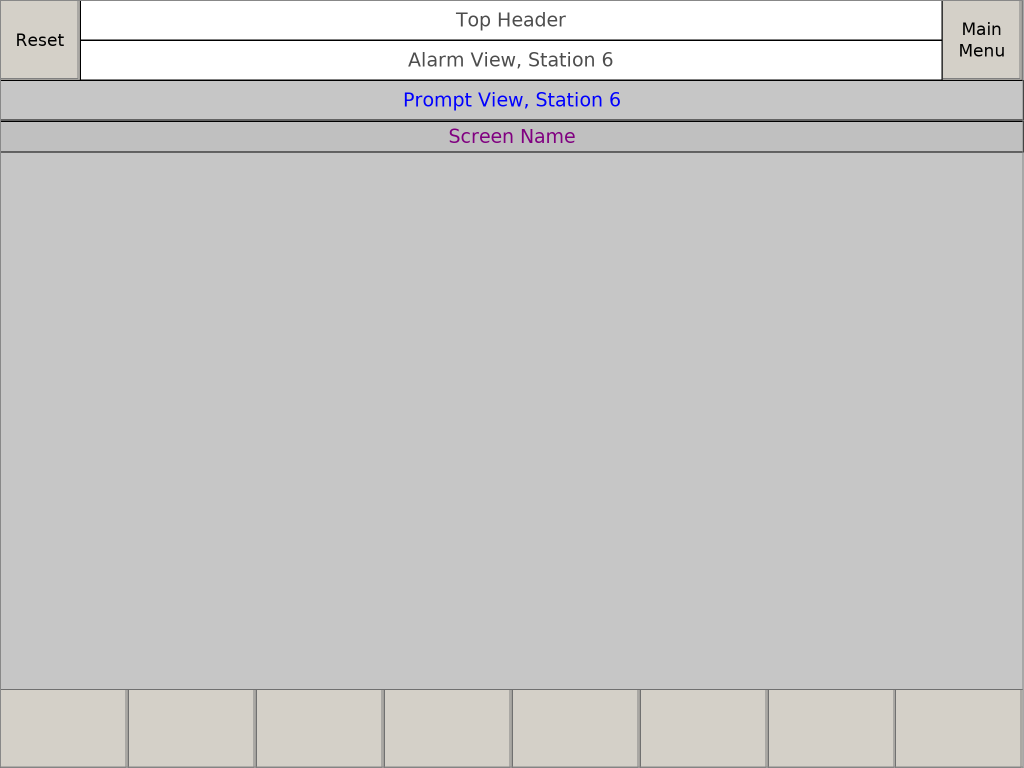
VISUALIZATION SS_91_Template  // 1024x768
    Button (0,0 80x80), "Reset"
    Button (942,0 80x80), "Main Menu"
        OnMouseClick: change screen: SS_10_MenuScreen
    Rectangle (0,80 1024x40), "Prompt View, Station 6", invisible if: GlobalHMIData.gHideDisplayElementPromptView.McEnabled, text list: 'Mc_Prompts', text index: GlobalHMIData.gNumActivePromptTextList[0]
    Rectangle (80,0 862x40), "Top Header"
    Button (0,689 128x80), invisible if: GlobalHMIData.gHideDisplayElementWarningView.S1Enabled
    Button (128,689 128x80)
    Button (256,689 128x80)
    Button (384,689 128x80)
    Button (512,689 128x80)
    Button (640,689 128x80)
    Button (768,689 128x80)
    Button (895,689 128x80)
    Rectangle (80,40 862x40), "Warning View, Machine", invisible if: GlobalHMIData.gHideDisplayElementWarningView.McEnabled, text list: 'Mc_Warnings', text index: GlobalHMIData.gNumActiveWarningTextList[0]
    Rectangle (80,40 862x40), "Warning View, Station 1", invisible if: GlobalHMIData.gHideDisplayElementWarningView.S1Enabled, text list: 'S1_Warnings', text index: GlobalHMIData.gNumActiveWarningTextList[1]
    Rectangle (80,40 862x40), "Warning View, Station 2", invisible if: GlobalHMIData.gHideDisplayElementWarningView.S2Enabled, text list: 'S2_Warnings', text index: GlobalHMIData.gNumActiveWarningTextList[2]
    Rectangle (80,40 862x40), "Warning View, Station 3", invisible if: GlobalHMIData.gHideDisplayElementWarningView.S3Enabled, text list: 'S3_Warnings', text index: GlobalHMIData.gNumActiveWarningTextList[3]
    Rectangle (80,40 862x40), "Warning View, Station 4", invisible if: GlobalHMIData.gHideDisplayElementWarningView.S4Enabled, text list: 'S4_Warnings', text index: GlobalHMIData.gNumActiveWarningTextList[4]
    Rectangle (80,40 862x40), "Warning View, Station 5", invisible if: GlobalHMIData.gHideDisplayElementWarningView.S5Enabled, text list: 'S5_Warnings', text index: GlobalHMIData.gNumActiveWarningTextList[5]
    Rectangle (80,40 862x40), "Warning View, Station 6", invisible if: GlobalHMIData.gHideDisplayElementWarningView.S6Enabled, text list: 'S6_Warnings', text index: GlobalHMIData.gNumActiveWarningTextList[6]
    Rectangle (80,40 862x40), "Alarm View, Machine", invisible if: GlobalHMIData.gHideDisplayElementAlarmView.McEnabled, text list: 'Mc_Alarms', text index: GlobalHMIData.gNumActiveAlarmTextList[0]
    Rectangle (80,40 862x40), "Alarm View, Station 1", invisible if: GlobalHMIData.gHideDisplayElementAlarmView.S1Enabled, text list: 'S1_Alarms', text index: GlobalHMIData.gNumActiveAlarmTextList[1]
    Rectangle (80,40 862x40), "Alarm View, Station 2", invisible if: GlobalHMIData.gHideDisplayElementAlarmView.S2Enabled, text list: 'S2_Alarms', text index: GlobalHMIData.gNumActiveAlarmTextList[2]
    Rectangle (80,40 862x40), "Alarm View, Station 3", invisible if: GlobalHMIData.gHideDisplayElementAlarmView.S3Enabled, text list: 'S3_Alarms', text index: GlobalHMIData.gNumActiveAlarmTextList[3]
    Rectangle (80,40 862x40), "Alarm View, Station 4", invisible if: GlobalHMIData.gHideDisplayElementAlarmView.S4Enabled, text list: 'S4_Alarms', text index: GlobalHMIData.gNumActiveAlarmTextList[4]
    Rectangle (80,40 862x40), "Alarm View, Station 5", invisible if: GlobalHMIData.gHideDisplayElementAlarmView.S5Enabled, text list: 'S5_Alarms', text index: GlobalHMIData.gNumActiveAlarmTextList[5]
    Rectangle (80,40 862x40), "Alarm View, Station 6", invisible if: GlobalHMIData.gHideDisplayElementAlarmView.S6Enabled, text list: 'S6_Alarms', text index: GlobalHMIData.gNumActiveAlarmTextList[6]
    Rectangle (0,80 1024x40), "Prompt View, Station 1", invisible if: GlobalHMIData.gHideDisplayElementPromptView.S1Enabled, text list: 'S1_Prompts', text index: GlobalHMIData.gNumActivePromptTextList[1]
    Rectangle (0,80 1024x40), "Prompt View, Station 2", invisible if: GlobalHMIData.gHideDisplayElementPromptView.S2Enabled, text list: 'S2_Prompts', text index: GlobalHMIData.gNumActivePromptTextList[2]
    Rectangle (0,80 1024x40), "Prompt View, Station 3", invisible if: GlobalHMIData.gHideDisplayElementPromptView.S3Enabled, text list: 'S3_Prompts', text index: GlobalHMIData.gNumActivePromptTextList[3]
    Rectangle (0,80 1024x40), "Prompt View, Station 4", invisible if: GlobalHMIData.gHideDisplayElementPromptView.S4Enabled, text list: 'S4_Prompts', text index: GlobalHMIData.gNumActivePromptTextList[4]
    Rectangle (0,80 1024x40), "Prompt View, Station 5", invisible if: GlobalHMIData.gHideDisplayElementPromptView.S5Enabled, text list: 'S5_Prompts', text index: GlobalHMIData.gNumActivePromptTextList[5]
    Rectangle (0,80 1024x40), "Prompt View, Station 6", invisible if: GlobalHMIData.gHideDisplayElementPromptView.S6Enabled, text list: 'S6_Prompts', text index: GlobalHMIData.gNumActivePromptTextList[6]
    Rectangle (0,121 1024x31), "Screen Name", invisible if: GlobalHMIData.gHideDisplayElementPromptView.S6Enabled, text list: 'ScreenNames', text index: GlobalHMIData.gScreenNumber
END_VISUALIZATION

(* stored: Version 1.1.0.1, ProductVersion 3.1.4024.12
   Visu SS_91_Template: Id {b17fde76-284b-401f-89cc-43a3764876ae} *)
